# EPICS substitutions: iocBoot/iocvirPV/DPU01.substitutions
file "../../db/virAi.template"{ pattern
{DPU,    num,    Temp}
{01,    0,    500}
{01,    1,    500}
{01,    2,    500}
{01,    3,    500}
{01,    4,    500}
{01,    5,    500}
{01,    6,    500}
{01,    7,    500}
{01,    8,    500}
{01,    9,    500}
{01,    10,    500}
{01,    11,    500}
{01,    12,    500}
{01,    13,    500}
{01,    14,    500}
{01,    15,    500}
{01,    16,    500}
{01,    17,    500}
{01,    18,    500}
{01,    19,    500}
{01,    20,    500}
{01,    21,    500}
{01,    22,    500}
{01,    23,    500}
{01,    24,    500}
{01,    25,    500}
{01,    26,    500}
{01,    27,    500}
{01,    28,    500}
{01,    29,    500}
{01,    30,    500}
{01,    31,    500}
{01,    32,    500}
{01,    33,    500}
{01,    34,    500}
{01,    35,    500}
{01,    36,    500}
{01,    37,    500}
{01,    38,    500}
{01,    39,    500}
{01,    40,    500}
{01,    41,    500}
{01,    42,    500}
{01,    43,    500}
{01,    44,    500}
{01,    45,    500}
{01,    46,    500}
{01,    47,    500}
{01,    48,    500}
{01,    49,    500}
{01,    50,    500}
{01,    51,    500}
{01,    52,    500}
{01,    53,    500}
{01,    54,    500}
{01,    55,    500}
{01,    56,    500}
{01,    57,    500}
{01,    58,    500}
{01,    59,    500}
{01,    60,    500}
{01,    61,    500}
{01,    62,    500}
{01,    63,    500}
{01,    64,    500}
{01,    65,    500}
{01,    66,    500}
{01,    67,    500}
{01,    68,    500}
{01,    69,    500}
{01,    70,    500}
{01,    71,    500}
{01,    72,    500}
{01,    73,    500}
{01,    74,    500}
{01,    75,    500}
{01,    76,    500}
{01,    77,    500}
{01,    78,    500}
{01,    79,    500}
{01,    80,    500}
{01,    81,    500}
{01,    82,    500}
{01,    83,    500}
{01,    84,    500}
{01,    85,    500}
{01,    86,    500}
{01,    87,    500}
{01,    88,    500}
{01,    89,    500}
{01,    90,    500}
{01,    91,    500}
{01,    92,    500}
{01,    93,    500}
{01,    94,    500}
{01,    95,    500}
{01,    96,    500}
{01,    97,    500}
{01,    98,    500}
{01,    99,    500}
{01,    100,    500}
{01,    101,    500}
{01,    102,    500}
{01,    103,    500}
{01,    104,    500}
{01,    105,    500}
{01,    106,    500}
{01,    107,    500}
{01,    108,    500}
{01,    109,    500}
{01,    110,    500}
{01,    111,    500}
{01,    112,    500}
{01,    113,    500}
{01,    114,    500}
{01,    115,    500}
{01,    116,    500}
{01,    117,    500}
{01,    118,    500}
{01,    119,    500}
{01,    120,    500}
{01,    121,    500}
{01,    122,    500}
{01,    123,    500}
{01,    124,    500}
{01,    125,    500}
{01,    126,    500}
{01,    127,    500}
{01,    128,    500}
{01,    129,    500}
{01,    130,    500}
{01,    131,    500}
{01,    132,    500}
{01,    133,    500}
{01,    134,    500}
{01,    135,    500}
{01,    136,    500}
{01,    137,    500}
{01,    138,    500}
{01,    139,    500}
{01,    140,    500}
{01,    141,    500}
{01,    142,    500}
{01,    143,    500}
{01,    144,    500}
{01,    145,    500}
{01,    146,    500}
{01,    147,    500}
{01,    148,    500}
{01,    149,    500}
{01,    150,    500}
{01,    151,    500}
{01,    152,    500}
{01,    153,    500}
{01,    154,    500}
{01,    155,    500}
{01,    156,    500}
{01,    157,    500}
{01,    158,    500}
{01,    159,    500}
{01,    160,    500}
{01,    161,    500}
{01,    162,    500}
{01,    163,    500}
{01,    164,    500}
{01,    165,    500}
{01,    166,    500}
{01,    167,    500}
{01,    168,    500}
{01,    169,    500}
{01,    170,    500}
{01,    171,    500}
{01,    172,    500}
{01,    173,    500}
{01,    174,    500}
{01,    175,    500}
{01,    176,    500}
{01,    177,    500}
{01,    178,    500}
{01,    179,    500}
{01,    180,    500}
{01,    181,    500}
{01,    182,    500}
{01,    183,    500}
{01,    184,    500}
{01,    185,    500}
{01,    186,    500}
{01,    187,    500}
{01,    188,    500}
{01,    189,    500}
{01,    190,    500}
{01,    191,    500}
{01,    192,    500}
{01,    193,    500}
{01,    194,    500}
{01,    195,    500}
{01,    196,    500}
{01,    197,    500}
{01,    198,    500}
{01,    199,    500}
}
